(* IEC 61131-3 sources: AXOpen/src/components.cognex.vision/ctrl/src/AxoDataman/v_6_0_0/TypeStructuresAndEnums, 16 files *)

(* ---- AxoDataman_AcquisitionControl.st ---- *)
NAMESPACE AXOpen.Components.Cognex.Vision.v_6_0_0_0
    TYPE
        AxoDataman_AcquisitionControl :
        STRUCT
            {#ix-set:AttributeName = "<#Trigger enable#>"}
            TriggerEnable : BOOL;
            {#ix-set:AttributeName = "<#Trigger#>"}
            Trigger : BOOL;
        END_STRUCT;
    END_TYPE
END_NAMESPACE

(* ---- AxoDataman_AcquisitionStatus.st ---- *)
NAMESPACE AXOpen.Cognex.Vision.v_6_0_0_0
    TYPE
        AxoDataman_AcquisitionStatus :
        STRUCT
            TriggerReady 		:	BOOL;
            TriggerAcknowledge 	:	BOOL;
            Acquiring 			:	BOOL;
            MissedAcquisition 	:	BOOL;
            TriggerID 			:	UINT;
        END_STRUCT;
    END_TYPE
END_NAMESPACE

(* ---- AxoDataman_Config.st ---- *)
NAMESPACE AXOpen.Components.Cognex.Vision.v_6_0_0_0
    TYPE
        {#ix-attr:[Container(Layout.Stack)]}
        {S7.extern=ReadWrite}
        AxoDataman_Config :
        STRUCT
            {#ix-set:AttributeName = "<#Continous reading#>"}
            ContinuousReading : BOOL := FALSE;
            {#ix-set:AttributeName = "<#Info time#>"}
            InfoTime : LTIME := LT#2S;
            {#ix-set:AttributeName = "<#Error time#>"}
            ErrorTime : LTIME := LT#5S;
            {#ix-set:AttributeName = "<#Task timeout#>"}
            TaskTimeout : LTIME := LT#50S;
            {#ix-set:AttributeName = "<#Result data size#>"}
            ResultDataSize : eAxoDataman_ResultDataSize := eAxoDataman_ResultDataSize#RESULT_DATA_SIZE_INVALID;
            {#ix-set:AttributeName = "<#User data size#>"}
            UserDataSize : eAxoDataman_UserDataSize := eAxoDataman_UserDataSize#USER_DATA_SIZE_INVALID;
        END_STRUCT;
    END_TYPE
END_NAMESPACE

(* ---- AxoDataman_Results.st ---- *)
NAMESPACE AXOpen.Components.Cognex.Vision.v_6_0_0_0
    TYPE
        AxoDataman_Results :
        STRUCT
            {#ix-set:AttributeName = "<#Id#>"}
            Id: UINT;
            {#ix-set:AttributeName = "<#Code#>"}
            Code: UINT;
            {#ix-set:AttributeName = "<#Extended#>"}
            Extended: UINT;
            {#ix-set:AttributeName = "<#Length#>"}
            Length : UINT;
        END_STRUCT;
    END_TYPE
END_NAMESPACE

(* ---- AxoDataman_ResultsControl.st ---- *)
NAMESPACE AXOpen.Components.Cognex.Vision.v_6_0_0_0
    TYPE
        AxoDataman_ResultsControl :
        STRUCT
            {#ix-set:AttributeName = "<#Enable results buffering#>"}
            EnableResultBuffering   :   BOOL;
            {#ix-set:AttributeName = "<#Results acknowledge#>"}
            ResultsAcknowledge      :   BOOL;
        END_STRUCT;
    END_TYPE
END_NAMESPACE

(* ---- AxoDataman_ResultsStatus.st ---- *)
NAMESPACE AXOpen.Cognex.Vision.v_6_0_0_0
    TYPE
        AxoDataman_ResultsStatus :
        STRUCT
            {#ix-set:AttributeName = "<#Decoding#>"}
            Decoding 			    :   BOOL;
            {#ix-set:AttributeName = "<#Decode complete#>"}
            DecodeComplete 		    :   BOOL;
            {#ix-set:AttributeName = "<#Results buffer overrun#>"}
            ResultsBufferOverrun    :   BOOL;
            {#ix-set:AttributeName = "<#Results available#>"}
            ResultsAvailable 	    :   BOOL;
            {#ix-set:AttributeName = "<#Error detected#>"}
            ErrorDetected 		    :   BOOL;
        END_STRUCT;
    END_TYPE
END_NAMESPACE

(* ---- AxoDataman_SignalStates.st ---- *)
NAMESPACE AXOpen.Cognex.Vision.v_6_0_0_0
    TYPE
        {#ix-set:AttributeName = "<#Signal states#>"}
        {#ix-attr:[Container(Layout.Wrap)]}
        AxoDataman_SignalStates :
        STRUCT
            {#ix-set:AttributeName = "<#Trigger enable#>"}
            TriggerEnable 			:	BOOL;
            {#ix-set:AttributeName = "<#Trigger#>"}
            Trigger					:	BOOL;

            {#ix-set:AttributeName = "<#Enable result buffering#>"}
            EnableResultBuffering	:	BOOL;
            {#ix-set:AttributeName = "<#Result acknowledge#>"}
            ResultsAcknowledge		:	BOOL;

            {#ix-set:AttributeName = "<#Trigger ready#>"}
            TriggerReady 		:	BOOL;
            {#ix-set:AttributeName = "<#Trigger acknowledge#>"}
            TriggerAcknowledge 	:	BOOL;
            {#ix-set:AttributeName = "<#Acquiring#>"}
            Acquiring 			:	BOOL;
            {#ix-set:AttributeName = "<#Missed acquisition#>"}
            MissedAcquisition 	:	BOOL;
            {#ix-set:AttributeName = "<#Trigger ID#>"}
            TriggerID 			:	UINT;

            {#ix-set:AttributeName = "<#Decoding#>"}
            Decoding 				:	BOOL;
            {#ix-set:AttributeName = "<#Decode complete#>"}
            DecodeComplete 			:	BOOL;
            {#ix-set:AttributeName = "<#Result buffer overrun#>"}
            ResultsBufferOverrun 	:	BOOL;
            {#ix-set:AttributeName = "<#Results available#>"}
            ResultsAvailable 		:	BOOL;
            {#ix-set:AttributeName = "<#Error detected#>"}
            ErrorDetected 			:	BOOL;

            {#ix-set:AttributeName = "<#Result ID#>"}
            ResultID 				:	UINT;
            {#ix-set:AttributeName = "<#Result code#>"}
            ResultCode  			:	UINT;
            {#ix-set:AttributeName = "<#Result extended#>"}
            ResultExtended  		:	UINT;
            {#ix-set:AttributeName = "<#Result length#>"}
            ResultLength  			:	UINT;
        END_STRUCT;
    END_TYPE
END_NAMESPACE

(* ---- AxoDataman_SoftEventControl.st ---- *)
NAMESPACE AXOpen.Cognex.Vision.v_6_0_0_0
    TYPE
        AxoDataman_SoftEventControl :
        STRUCT
            {#ix-set:AttributeName = "<#Train code#>"}
            TrainCode 						:   BOOL;
            {#ix-set:AttributeName = "<#Train match string#>"}
            TrainMatchString 				:   BOOL;
            {#ix-set:AttributeName = "<#Train focus#>"}
            TrainFocus 						:   BOOL;
            {#ix-set:AttributeName = "<#Train brightness#>"}
            TrainBrightness 				:   BOOL;
            {#ix-set:AttributeName = "<#Untrain#>"}
            Untrain 						:   BOOL;
            {#ix-set:AttributeName = "<#Execute DMCC#>"}
            ExecuteDMCC 					:   BOOL;
            {#ix-attr:[CompilerOmits()]}
            Reserved06 						:   BOOL;
            {#ix-set:AttributeName = "<#Decoding#>"}
            SetMatchString 					:   BOOL;
        END_STRUCT;
    END_TYPE
END_NAMESPACE

(* ---- AxoDataman_SoftEventStatus.st ---- *)
NAMESPACE AXOpen.Components.Cognex.Vision.v_6_0_0_0
    TYPE
        AxoDataman_SoftEventStatus :
        STRUCT
            {#ix-set:AttributeName = "<#Train code acknowledge#>"}
            TrainCodeAcknowledge 			:   BOOL;
            {#ix-set:AttributeName = "<#Train match string acknowledge#>"}
            TrainMatchStringAcknowledge 	:   BOOL;
            {#ix-set:AttributeName = "<#Train focus acknowledge#>"}
            TrainFocusAcknowledge 			:   BOOL;
            {#ix-set:AttributeName = "<#Train brightness acknowledge#>"}
            TrainBrightnessAcknowledge  	:   BOOL;
            {#ix-set:AttributeName = "<#Untrain acknowledge#>"}
            UntrainAcknowledge  			:   BOOL;
            {#ix-set:AttributeName = "<#Execute DMCC acknowledge#>"}
            ExecuteDMCCAcknowledge 			:   BOOL;
            {#ix-attr:[CompilerOmits()]}
            Reserved06 						:   BOOL;
            {#ix-set:AttributeName = "<#Set match string acknowledge#>"}
            SetMatchStringAcknowledge  		:   BOOL;
        END_STRUCT;
    END_TYPE
END_NAMESPACE

(* ---- AxoDataman_User.st ---- *)
NAMESPACE AXOpen.Cognex.Vision.v_6_0_0_0
    TYPE
        AxoDataman_User :
        STRUCT
            {#ix-set:AttributeName = "<#Option#>"}
            Option : UINT;
            {#ix-set:AttributeName = "<#Length#>"}
            Length : UINT;
        END_STRUCT;
    END_TYPE
END_NAMESPACE

(* ---- eAxoDataman_ResultDataSize.st ---- *)
NAMESPACE AXOpen.Components.Cognex.Vision.v_6_0_0_0
    TYPE PUBLIC
        eAxoDataman_ResultDataSize : INT
        (
            RESULT_DATA_SIZE_INVALID := 0,
            RESULT_DATA_16B := 16,
            RESULT_DATA_32B := 32,
            RESULT_DATA_64B := 64,
            RESULT_DATA_128B := 128,
            RESULT_DATA_246B := 246
         ) := RESULT_DATA_64B;
    END_TYPE
END_NAMESPACE

(* ---- eAxoDataman_UserDataSize.st ---- *)
NAMESPACE AXOpen.Cognex.Vision.v_6_0_0_0
    TYPE PUBLIC
        eAxoDataman_UserDataSize : INT
        (
            USER_DATA_SIZE_INVALID := 0,
            USER_DATA_16B := 16,
            USER_DATA_32B := 32,
            USER_DATA_64B := 64,
            USER_DATA_128B := 128,
            USER_DATA_250B := 250
         ) := USER_DATA_64B;
    END_TYPE
END_NAMESPACE

(* ---- AxoDataman_HWIDs.st ---- *)
NAMESPACE AXOpen.Components.Cognex.Vision.v_6_0_0_0
    {#ix-attr:[Container(Layout.Stack)]}
    {S7.extern=ReadWrite}
    CLASS PUBLIC AxoDataman_HWIDs
        VAR PUBLIC
            {#ix-set:AttributeName = "<#Hardware ID of the device#>"}
            HW_Device               :  UINT;
            {#ix-set:AttributeName = "<#Hardware ID of the 'AcquisitionControl' submodule#>"}
            HwIdAcquisitionControl  :   UINT;
            {#ix-set:AttributeName = "<#Hardware ID of the 'AcquisitionStatus' submodule#>"}
            HwIdAcquisitionStatus   :   UINT;
            {#ix-set:AttributeName = "<#Hardware ID of the 'ResultsControl' submodule#>"}
            HwIdResultsControl      :   UINT;
            {#ix-set:AttributeName = "<#Hardware ID of the 'ResultsStatus' submodule#>"}
            HwIdResultsStatus       :   UINT;
            {#ix-set:AttributeName = "<#Hardware ID of the 'SoftEventControl' submodule#>"}
            HwIdSoftEventControl    :   UINT;
            {#ix-set:AttributeName = "<#Hardware ID of the 'UserData' submodule#>"}
            HwIdUserData            :   UINT;
            {#ix-set:AttributeName = "<#Hardware ID of the 'ResultData' submodule#>"}
            HwIdResultData          :   UINT;
        END_VAR
    END_CLASS
END_NAMESPACE

(* ---- AxoDataman_ResultData.st ---- *)
NAMESPACE AXOpen.Cognex.Vision.v_6_0_0_0
    CLASS PUBLIC AxoDataman_ResultData EXTENDS AXOpen.Core.AxoByteArray
        VAR PUBLIC
            Data : ARRAY [0..245] OF BYTE;
        END_VAR
    END_CLASS
END_NAMESPACE

(* ---- AxoDataman_Status.st ---- *)
USING AXOpen.Components.Core;
NAMESPACE AXOpen.Components.Cognex.Vision.v_6_0_0_0
    {#ix-attr:[Container(Layout.Stack)]}
    {S7.extern=ReadWrite}
    CLASS AxoDataman_Status EXTENDS AXOpen.Components.Abstractions.AxoComponent_Status
        VAR PUBLIC
            // {#ix-attr:[Container(Layout.Wrap)]}
            // ResultDataSize : eAxoDataman_ResultDataSize := eAxoDataman_ResultDataSize#RESULT_DATA_SIZE_INVALID;
            // {#ix-attr:[CompilerOmits()]}
            // UserDataSize : eAxoDataman_UserDataSize := eAxoDataman_UserDataSize#USER_DATA_SIZE_INVALID;
        END_VAR
    END_CLASS
END_NAMESPACE

(* ---- AxoDataman_UserData.st ---- *)
NAMESPACE AXOpen.Components.Cognex.Vision.v_6_0_0_0
    CLASS PUBLIC AxoDataman_UserData EXTENDS AXOpen.Core.AxoByteArray
        VAR PUBLIC
            Data : ARRAY [0..249] OF BYTE;
        END_VAR
    END_CLASS
END_NAMESPACE
